FUNCTION Func : WORD
VAR_INPUT
	a:WORD;
	b:WORD;
END_VAR
VAR
	c:WORD;
END_VAR

c:=a+b;
Func:=c;
RETURN;

END_FUNCTION

(* stored: Version 1.1.0.1, ProductVersion 3.1.4024.12
   POU Func: Id {be6bc712-9ba6-4b33-9677-cb41ac6cdef4}, SpecialFunc None *)
